FUNCTION F_EndsWith : BOOL
VAR_INPUT
    s      : STRING;
    suffix : STRING;
END_VAR

END_FUNCTION

(* stored: Version 1.1.0.1
   POU F_EndsWith: Id {1f7dac19-833e-4d40-a03c-3c7468787a8b}, SpecialFunc None *)
